// This function has been automatically generated from the project information.
{attribute 'signature_flag' := '1073741824'}
{attribute 'TcGenerated'}
{attribute 'no-analysis'}
FUNCTION F_GetTitle : WSTRING
VAR_INPUT
	
END_VAR

F_GetTitle := "FsGenerics";

END_FUNCTION

(* stored: Version 1.1.0.1
   POU F_GetTitle: Id {bbf4f11a-e56d-47fc-93bc-530d60e81f46}, SpecialFunc None *)
